RoboDK station: Table with plates.rdk

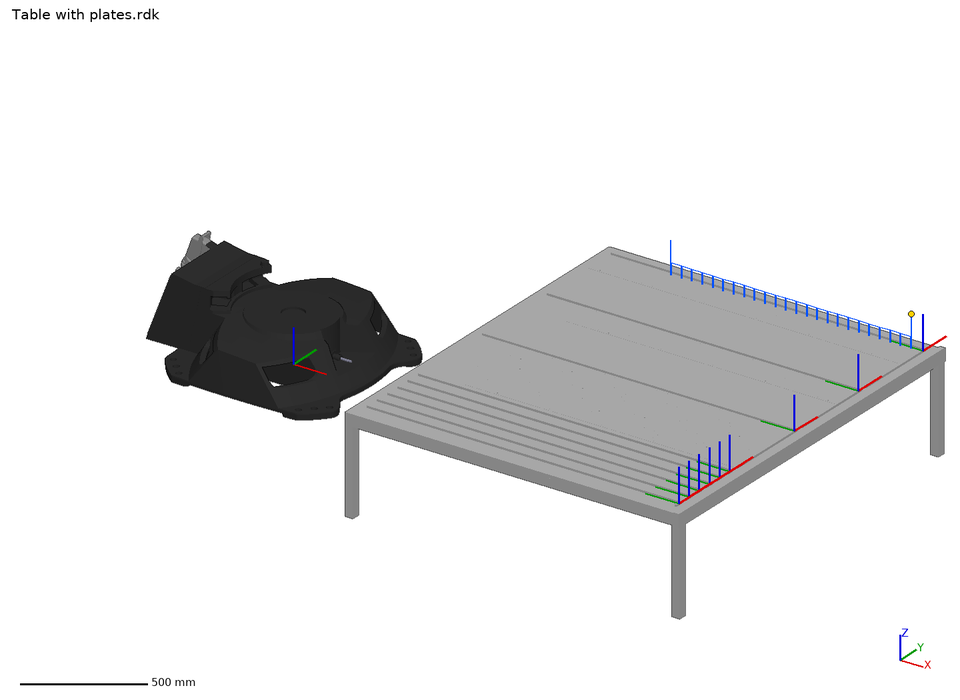
[picture v0: the station drawn from its stored meshes, robots at their saved joint values, targets as dots, program paths as lines]
Station Table with plates (saved by RoboDK 5.2.3). Poses are relative to the parent item; angles as X-Y-Z fixed-axis rotations.
  - frame KUKA KR 210 R2700 extra Base at (0, 1000, 0) mm
    - robot KUKA KR 210 R2700 extra: 6 axes, payload 210 kg, reach 2696 mm, repeatability 0.06 mm, weight 1068 kg
        joint limits [-185, -140, -120, -350, -125, -350] to [185, -5, 155, 350, 125, 350]; home [0, -90, 90, 0, 0, 0]; saved at [30.44, -87.596, 137.193, -142.344, 56.026, 156.673]
      - tool Spindle, TCP at (278.6, 0, 88) mm, rotated rx 0 ry 90 rz 0 deg, size 85 x 346.5 x 128 mm
  - object Table at (1700, 300, 400) mm, rotated rx 0 ry 0 rz 90 deg, size 1820 x 1605 x 465 mm
  - frame Plate 1 at (2490, 1750, 455) mm, rotated rx 0 ry 0 rz 90 deg
  - frame Plate 2 at (2490, 1310, 455) mm, rotated rx 0 ry 0 rz 90 deg
  - frame Plate 3 at (2490, 870, 455) mm, rotated rx 0 ry 0 rz 90 deg
  - frame Stringer 1 at (2490, 430, 455) mm, rotated rx 0 ry 0 rz 90 deg
  - frame Stringer 2 at (2490, 360, 455) mm, rotated rx 0 ry 0 rz 90 deg
  - frame Stringer 3 at (2490, 290, 455) mm, rotated rx 0 ry 0 rz 90 deg
  - frame Stringer 4 at (2490, 220, 455) mm, rotated rx 0 ry 0 rz 90 deg
  - frame Stringer 5 at (2490, 150, 455) mm, rotated rx 0 ry 0 rz 90 deg
  - frame Stringer 6 at (2490, 80, 455) mm, rotated rx 0 ry 0 rz 90 deg
  - object WB1_Stringer_B1 at (2490, 430, 455) mm, rotated rx 0 ry 0 rz 90 deg
  - program Path1 (84 instructions, listed below)
  - object WB1_sheet_A at (1740, 1762.91, 455) mm, rotated rx 0 ry 0 rz 180 deg, size 1500 x 148.4 x 0.8 mm, geometry from WB1_sheet_A.stl
  - object WB1_sheet_A at (2490, 1750, 455) mm, rotated rx 0 ry 0 rz 90 deg
  - machining project Path1 settings: rotZ(0) | rotX(0)*rotY(0) | rotz(0) | onStart | onPathStart | onApproach | onPoint | onRetract | onFinish | SetRPM(%1) | SetTool(%1) | Extruder(%1) | default | default | OutOnMov(%1) | OutOffMov(%1) | onPathFinish | M_RunCode(%1)
  - object WB1_sheet_B at (1840, 1235.8, 455) mm, rotated rx 0 ry 0 rz 180 deg, size 1300 x 148.4 x 0.8 mm, geometry from WB1_sheet_B.stl
  - object WB1_sheet_B at (2490, 1310, 455) mm, rotated rx 0 ry 0 rz 90 deg
  - object WB1_sheet_c1 at (1740, 670, 455.8) mm, rotated rx 180 ry 0 rz 180 deg, size 1500 x 400 x 0.8 mm, geometry from WB1_sheet_c1.stl
  - object WB1_sheet_C1 at (2490, 870, 455) mm, rotated rx 0 ry 0 rz 90 deg
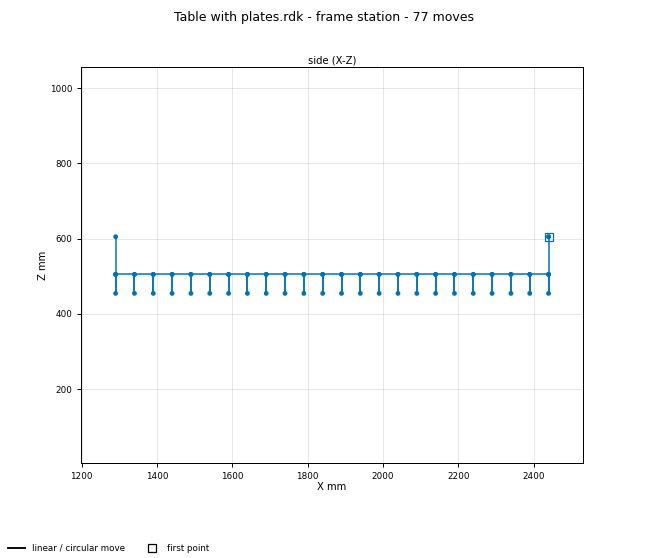
[picture p0: tool path of Table with plates.rdk in frame station, 77 of 77 moves have a stored position in this frame; points joined in program order, loops and branches not executed]

--- program Path1 (robot KUKA KR 210 R2700 extra) ---
  Smooth(1)
  Set speed (1000.0 mm/s)
  Set Ref.: Plate 1
  Set Tool: Spindle
  Show Spindle
  MoveJ 1 to (-10, 50, 150) mm, rotated rx 180 ry 0 rz 90 deg; joints [15.185, -44.385, 72.177, -149.797, 31.377, 153.575]
  MoveL 2 to (-10, 50, 150) mm, rotated rx 180 ry 0 rz 90 deg; joints [15.185, -44.385, 72.177, -149.797, 31.377, 153.575]
  MoveL 3 to (-10, 50, 50) mm, rotated rx 180 ry 0 rz 90 deg; joints [15.185, -41.687, 72.86, -152.33, 34.337, 156.589]
  MoveL 4 to (-10, 50, 50) mm, rotated rx 180 ry 0 rz 90 deg; joints [15.185, -41.687, 72.86, -152.33, 34.337, 156.589]
  Set speed (50.0 mm/s)
  MoveL 5 to (-10, 50, -0.5) mm, rotated rx 180 ry 0 rz 90 deg; joints [15.185, -40.232, 73.041, -153.394, 35.793, 157.888]
  MoveL 6 to (-10, 50, 50) mm, rotated rx 180 ry 0 rz 90 deg; joints [15.185, -41.687, 72.86, -152.33, 34.337, 156.589]
  MoveL 7 to (-10, 100, 50) mm, rotated rx 180 ry 0 rz 90 deg; joints [15.531, -43.734, 76.644, -152.91, 36.014, 157.523]
  MoveL 8 to (-10, 100, -0.5) mm, rotated rx 180 ry 0 rz 90 deg; joints [15.531, -42.236, 76.822, -153.914, 37.513, 158.776]
  MoveL 9 to (-10, 100, 50) mm, rotated rx 180 ry 0 rz 90 deg; joints [15.531, -43.734, 76.644, -152.91, 36.014, 157.523]
  MoveL 10 to (-10, 150, 50) mm, rotated rx -180 ry 0 rz 90 deg; joints [15.893, -45.709, 80.274, -153.349, 37.627, 158.323]
  MoveL 11 to (-10, 150, -0.5) mm, rotated rx -180 ry 0 rz 90 deg; joints [15.893, -44.168, 80.451, -154.305, 39.169, 159.543]
  MoveL 12 to (-10, 150, 50) mm, rotated rx -180 ry 0 rz 90 deg; joints [15.893, -45.709, 80.274, -153.349, 37.627, 158.323]
  MoveL 13 to (-10, 200, 50) mm, rotated rx 180 ry 0 rz 90 deg; joints [16.272, -47.624, 83.771, -153.671, 39.181, 159.014]
  MoveL 14 to (-10, 200, -0.5) mm, rotated rx -180 ry 0 rz 90 deg; joints [16.272, -46.036, 83.946, -154.588, 40.767, 160.211]
  MoveL 15 to (-10, 200, 50) mm, rotated rx 180 ry 0 rz 90 deg; joints [16.272, -47.624, 83.771, -153.671, 39.181, 159.014]
  MoveL 16 to (-10, 250, 50) mm, rotated rx 180 ry 0 rz 90 deg; joints [16.669, -49.486, 87.149, -153.893, 40.681, 159.613]
  MoveL 17 to (-10, 250, -0.5) mm, rotated rx 180 ry 0 rz 90 deg; joints [16.669, -47.851, 87.324, -154.779, 42.312, 160.796]
  MoveL 18 to (-10, 250, 50) mm, rotated rx 180 ry 0 rz 90 deg; joints [16.669, -49.486, 87.149, -153.893, 40.681, 159.613]
  MoveL 19 to (-10, 300, 50) mm, rotated rx 180 ry 0 rz 90 deg; joints [17.086, -51.303, 90.422, -154.026, 42.132, 160.136]
  MoveL 20 to (-10, 300, -0.5) mm, rotated rx -180 ry 0 rz 90 deg; joints [17.086, -49.617, 90.596, -154.887, 43.811, 161.313]
  MoveL 21 to (-10, 300, 50) mm, rotated rx 180 ry 0 rz 90 deg; joints [17.086, -51.303, 90.422, -154.026, 42.132, 160.136]
  MoveL 22 to (-10, 350, 50) mm, rotated rx -180 ry 0 rz 90 deg; joints [17.523, -53.081, 93.599, -154.082, 43.538, 160.593]
  MoveL 23 to (-10, 350, -0.5) mm, rotated rx 180 ry 0 rz 90 deg; joints [17.523, -51.342, 93.775, -154.923, 45.265, 161.771]
  MoveL 24 to (-10, 350, 50) mm, rotated rx -180 ry 0 rz 90 deg; joints [17.523, -53.081, 93.599, -154.082, 43.538, 160.593]
  MoveL 25 to (-10, 400, 50) mm, rotated rx 180 ry 0 rz 90 deg; joints [17.982, -54.825, 96.691, -154.065, 44.901, 160.993]
  MoveL 26 to (-10, 400, -0.5) mm, rotated rx 180 ry 0 rz 90 deg; joints [17.982, -53.031, 96.868, -154.892, 46.679, 162.177]
  MoveL 27 to (-10, 400, 50) mm, rotated rx 180 ry 0 rz 90 deg; joints [17.982, -54.825, 96.691, -154.065, 44.901, 160.993]
  MoveL 28 to (-10, 450, 50) mm, rotated rx -180 ry 0 rz 90 deg; joints [18.465, -56.54, 99.705, -153.983, 46.224, 161.341]
  MoveL 29 to (-10, 450, -0.5) mm, rotated rx 180 ry 0 rz 90 deg; joints [18.465, -54.688, 99.883, -154.798, 48.056, 162.538]
  MoveL 30 to (-10, 450, 50) mm, rotated rx -180 ry 0 rz 90 deg; joints [18.465, -56.54, 99.705, -153.983, 46.224, 161.341]
  MoveL 31 to (-10, 500, 50) mm, rotated rx -180 ry 0 rz 90 deg; joints [18.973, -58.231, 102.646, -153.837, 47.508, 161.642]
  MoveL 32 to (-10, 500, -0.5) mm, rotated rx 180 ry 0 rz 90 deg; joints [18.973, -56.316, 102.827, -154.644, 49.396, 162.859]
  MoveL 33 to (-10, 500, 50) mm, rotated rx -180 ry 0 rz 90 deg; joints [18.973, -58.231, 102.646, -153.837, 47.508, 161.642]
  MoveL 34 to (-10, 550, 50) mm, rotated rx -180 ry 0 rz 90 deg; joints [19.51, -59.901, 105.521, -153.631, 48.757, 161.902]
  MoveL 35 to (-10, 550, -0.5) mm, rotated rx 180 ry 0 rz 90 deg; joints [19.51, -57.92, 105.704, -154.434, 50.703, 163.144]
  MoveL 36 to (-10, 550, 50) mm, rotated rx -180 ry 0 rz 90 deg; joints [19.51, -59.901, 105.521, -153.631, 48.757, 161.902]
  MoveL 37 to (-10, 600, 50) mm, rotated rx 180 ry 0 rz 90 deg; joints [20.076, -61.554, 108.334, -153.366, 49.97, 162.122]
  MoveL 38 to (-10, 600, -0.5) mm, rotated rx -180 ry 0 rz 90 deg; joints [20.076, -59.502, 108.52, -154.168, 51.978, 163.395]
  MoveL 39 to (-10, 600, 50) mm, rotated rx 180 ry 0 rz 90 deg; joints [20.076, -61.554, 108.334, -153.366, 49.97, 162.122]
  MoveL 40 to (-10, 650, 50) mm, rotated rx -180 ry 0 rz 90 deg; joints [20.674, -63.193, 111.089, -153.041, 51.149, 162.304]
  MoveL 41 to (-10, 650, -0.5) mm, rotated rx 180 ry 0 rz 90 deg; joints [20.674, -61.066, 111.279, -153.845, 53.221, 163.616]
  MoveL 42 to (-10, 650, 50) mm, rotated rx -180 ry 0 rz 90 deg; joints [20.674, -63.193, 111.089, -153.041, 51.149, 162.304]
  MoveL 43 to (-10, 700, 50) mm, rotated rx 180 ry 0 rz 90 deg; joints [21.308, -64.821, 113.789, -152.658, 52.295, 162.451]
  MoveL 44 to (-10, 700, -0.5) mm, rotated rx 180 ry 0 rz 90 deg; joints [21.308, -62.614, 113.983, -153.467, 54.435, 163.806]
  MoveL 45 to (-10, 700, 50) mm, rotated rx 180 ry 0 rz 90 deg; joints [21.308, -64.821, 113.789, -152.658, 52.295, 162.451]
  MoveL 46 to (-10, 750, 50) mm, rotated rx 180 ry 0 rz 90 deg; joints [21.98, -66.442, 116.438, -152.214, 53.408, 162.562]
  MoveL 47 to (-10, 750, -0.5) mm, rotated rx -180 ry 0 rz 90 deg; joints [21.98, -64.15, 116.637, -153.031, 55.62, 163.969]
  MoveL 48 to (-10, 750, 50) mm, rotated rx 180 ry 0 rz 90 deg; joints [21.98, -66.442, 116.438, -152.214, 53.408, 162.562]
  MoveL 49 to (-10, 800, 50) mm, rotated rx -180 ry 0 rz 90 deg; joints [22.693, -68.059, 119.037, -151.709, 54.488, 162.638]
  MoveL 50 to (-10, 800, -0.5) mm, rotated rx 180 ry 0 rz 90 deg; joints [22.693, -65.675, 119.241, -152.537, 56.776, 164.104]
  MoveL 51 to (-10, 800, 50) mm, rotated rx -180 ry 0 rz 90 deg; joints [22.693, -68.059, 119.037, -151.709, 54.488, 162.638]
  MoveL 52 to (-10, 850, 50) mm, rotated rx 180 ry 0 rz 90 deg; joints [23.452, -69.675, 121.589, -151.138, 55.536, 162.678]
  MoveL 53 to (-10, 850, -0.5) mm, rotated rx -180 ry 0 rz 90 deg; joints [23.452, -67.192, 121.799, -151.98, 57.904, 164.212]
  MoveL 54 to (-10, 850, 50) mm, rotated rx 180 ry 0 rz 90 deg; joints [23.452, -69.675, 121.589, -151.138, 55.536, 162.678]
  MoveL 55 to (-10, 900, 50) mm, rotated rx 180 ry 0 rz 90 deg; joints [24.259, -71.293, 124.096, -150.5, 56.552, 162.68]
  MoveL 56 to (-10, 900, -0.5) mm, rotated rx 180 ry 0 rz 90 deg; joints [24.259, -68.705, 124.312, -151.36, 59.004, 164.291]
  MoveL 57 to (-10, 900, 50) mm, rotated rx 180 ry 0 rz 90 deg; joints [24.259, -71.293, 124.096, -150.5, 56.552, 162.68]
  MoveL 58 to (-10, 950, 50) mm, rotated rx 180 ry 0 rz 90 deg; joints [25.121, -72.918, 126.557, -149.79, 57.535, 162.644]
  MoveL 59 to (-10, 950, -0.5) mm, rotated rx 180 ry 0 rz 90 deg; joints [25.121, -70.215, 126.781, -150.67, 60.075, 164.343]
  MoveL 60 to (-10, 950, 50) mm, rotated rx 180 ry 0 rz 90 deg; joints [25.121, -72.918, 126.557, -149.79, 57.535, 162.644]
  MoveL 61 to (-10, 1000, 50) mm, rotated rx 180 ry 0 rz 90 deg; joints [26.041, -74.552, 128.975, -149.004, 58.484, 162.566]
  MoveL 62 to (-10, 1000, -0.5) mm, rotated rx 180 ry 0 rz 90 deg; joints [26.041, -71.725, 129.207, -149.909, 61.119, 164.364]
  MoveL 63 to (-10, 1000, 50) mm, rotated rx 180 ry 0 rz 90 deg; joints [26.041, -74.552, 128.975, -149.004, 58.484, 162.566]
  MoveL 64 to (-10, 1050, 50) mm, rotated rx 180 ry 0 rz 90 deg; joints [27.027, -76.2, 131.35, -148.135, 59.401, 162.442]
  MoveL 65 to (-10, 1050, -0.5) mm, rotated rx 180 ry 0 rz 90 deg; joints [27.027, -73.239, 131.59, -149.069, 62.133, 164.353]
  MoveL 66 to (-10, 1050, 50) mm, rotated rx 180 ry 0 rz 90 deg; joints [27.027, -76.2, 131.35, -148.135, 59.401, 162.442]
  MoveL 67 to (-10, 1100, 50) mm, rotated rx 180 ry 0 rz 90 deg; joints [28.083, -77.866, 133.681, -147.177, 60.283, 162.268]
  MoveL 68 to (-10, 1100, -0.5) mm, rotated rx 180 ry 0 rz 90 deg; joints [28.083, -74.76, 133.931, -148.144, 63.119, 164.307]
  MoveL 69 to (-10, 1100, 50) mm, rotated rx 180 ry 0 rz 90 deg; joints [28.083, -77.866, 133.681, -147.177, 60.283, 162.268]
  MoveL 70 to (-10, 1150, 50) mm, rotated rx 180 ry 0 rz 90 deg; joints [29.219, -79.554, 135.968, -146.123, 61.131, 162.04]
  MoveL 71 to (-10, 1150, -0.5) mm, rotated rx 180 ry 0 rz 90 deg; joints [29.219, -76.29, 136.229, -147.128, 64.076, 164.224]
  MoveL 72 to (-10, 1150, 50) mm, rotated rx 180 ry 0 rz 90 deg; joints [29.219, -79.554, 135.968, -146.123, 61.131, 162.04]
  MoveL 73 to (-10, 1200, 50) mm, rotated rx -180 ry 0 rz 90 deg; joints [30.44, -81.271, 138.21, -144.963, 61.944, 161.749]
  MoveL 74 to (-10, 1200, -0.5) mm, rotated rx 180 ry 0 rz 90 deg; joints [30.44, -77.833, 138.484, -146.013, 65.003, 164.098]
  MoveL 75 to (-10, 1200, 50) mm, rotated rx -180 ry 0 rz 90 deg; joints [30.44, -81.271, 138.21, -144.963, 61.944, 161.749]
  Set speed (1000.0 mm/s)
  MoveL 76 to (-10, 1200, 50) mm, rotated rx -180 ry 0 rz 90 deg; joints [30.44, -81.271, 138.21, -144.963, 61.944, 161.749]
  MoveL 77 to (-10, 1200, 150) mm, rotated rx 180 ry 0 rz 90 deg; joints [30.44, -87.596, 137.193, -142.344, 56.026, 156.673]
